// TIA Portal V15 export
// export: Created 2018-02-08T09:49:59.3125561Z, ExportSetting None, DisplayName Totally Integrated Automation Portal, DisplayVersion V15, DisplayName TIA Portal Openness, DisplayVersion V15, DisplayName TIA Portal Teamcenter Gateway, DisplayVersion V15, DisplayName SINAMICS Startdrive Advanced, DisplayVersion V15, DisplayName G110M, G120, G120C, G120D, G120P, DisplayVersion V15, DisplayName G130, G150, S120, S150, SINAMICS MV, DisplayVersion V15, DisplayName STEP 7 Professional, DisplayVersion V15, DisplayName WinCC Professional, DisplayVersion V15, DisplayName SIMATIC Visualization Architect, DisplayVersion V15
FUNCTION_BLOCK "Workshop1"   // FB2, LAD
{ S7_Optimized_Access := 'TRUE' }
// stored: AutoNumber false, MemoryReserve 100, SetENOAutomatically False
BEGIN

REGION Network 1
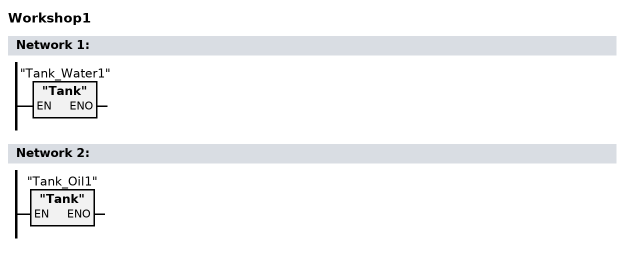
   RUNG wire#powerrail
      "Tank_Water1"()
   END_RUNG
   // the same network as SCL:
   "Tank_Water1"();   // "Tank"
END_REGION

REGION Network 2
   RUNG wire#powerrail
      "Tank_Oil1"()
   END_RUNG
   // the same network as SCL:
   "Tank_Oil1"();   // "Tank"
END_REGION
END_FUNCTION_BLOCK
